// Mitsubishi GX Works2 project: YYYY   PLC: Q02/Q02H

PROGRAM MAIN
VAR
  시작 : BOOL;
END_VAR
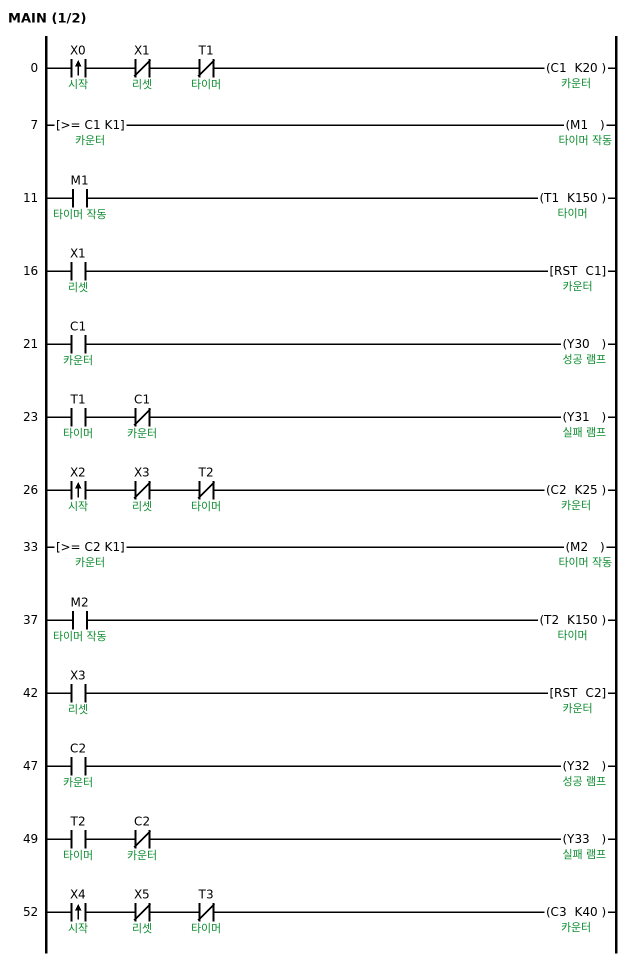
0     LDP     X0  ; 시작
      ANI     X1  ; 리셋
      ANI     T1  ; 타이머
      OUT     C1 K20  ; 카운터
7     LD>=    C1 K1  ; 카운터
      OUT     M1  ; 타이머 작동
11    LD      M1  ; 타이머 작동
      OUT     T1 K150  ; 타이머
16    LD      X1  ; 리셋
      RST     C1  ; 카운터
21    LD      C1  ; 카운터
      OUT     Y30  ; 성공 램프
23    LD      T1  ; 타이머
      ANI     C1  ; 카운터
      OUT     Y31  ; 실패 램프
26    LDP     X2  ; 시작
      ANI     X3  ; 리셋
      ANI     T2  ; 타이머
      OUT     C2 K25  ; 카운터
33    LD>=    C2 K1  ; 카운터
      OUT     M2  ; 타이머 작동
37    LD      M2  ; 타이머 작동
      OUT     T2 K150  ; 타이머
42    LD      X3  ; 리셋
      RST     C2  ; 카운터
47    LD      C2  ; 카운터
      OUT     Y32  ; 성공 램프
49    LD      T2  ; 타이머
      ANI     C2  ; 카운터
      OUT     Y33  ; 실패 램프
52    LDP     X4  ; 시작
      ANI     X5  ; 리셋
      ANI     T3  ; 타이머
      OUT     C3 K40  ; 카운터
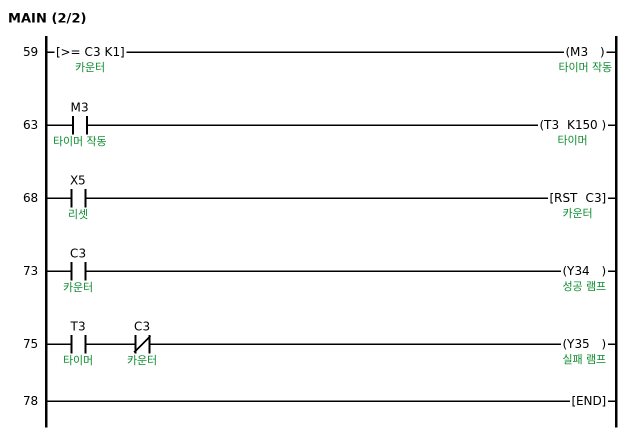
59    LD>=    C3 K1  ; 카운터
      OUT     M3  ; 타이머 작동
63    LD      M3  ; 타이머 작동
      OUT     T3 K150  ; 타이머
68    LD      X5  ; 리셋
      RST     C3  ; 카운터
73    LD      C3  ; 카운터
      OUT     Y34  ; 성공 램프
75    LD      T3  ; 타이머
      ANI     C3  ; 카운터
      OUT     Y35  ; 실패 램프
78    END
END_PROGRAM
